(* CODESYS project 96lPixBadAppleControlWin.project

Project tree, tasks and I/O mapping:
  Device : CODESYS Control Win V3, 3S - Smart Software Solutions GmbH, order no. 305021, version 3.5.10.40
    application Application
      libraries: Standard, * (System); CAA File, 3.5.9.0 (CAA Technical Workgroup)
      task MainTask (cyclic, interval t#20ms, priority 1) calls PLC_PRG
      task VISU_TASK (cyclic, interval 100 ms, priority 31) calls VisuElems.Visu_Prg
      program PLC_PRG [ST]
      visualisation Visualization
      data type bigStruct
      data type bigUnion
      data type smallUnion
  visualisation LPixboard
  text list GlobalTextList
*)

// Device/Application/bigStruct
TYPE bigStruct :
STRUCT
	structLine0: ARRAY [0..11] OF BYTE;
	structLine1: ARRAY [0..11] OF BYTE;
	structLine2: ARRAY [0..11] OF BYTE;
	structLine3: ARRAY [0..11] OF BYTE;
	structLine4: ARRAY [0..11] OF BYTE;
	structLine5: ARRAY [0..11] OF BYTE;
	structLine6: ARRAY [0..11] OF BYTE;
	structLine7: ARRAY [0..11] OF BYTE;
	structLine8: ARRAY [0..11] OF BYTE;
	structLine9: ARRAY [0..11] OF BYTE;
	structLine10: ARRAY [0..11] OF BYTE;
	structLine11: ARRAY [0..11] OF BYTE;
	structLine12: ARRAY [0..11] OF BYTE;
	structLine13: ARRAY [0..11] OF BYTE;
	structLine14: ARRAY [0..11] OF BYTE;
	structLine15: ARRAY [0..11] OF BYTE;
	structLine16: ARRAY [0..11] OF BYTE;
	structLine17: ARRAY [0..11] OF BYTE;
	structLine18: ARRAY [0..11] OF BYTE;
	structLine19: ARRAY [0..11] OF BYTE;
	structLine20: ARRAY [0..11] OF BYTE;
	structLine21: ARRAY [0..11] OF BYTE;
	structLine22: ARRAY [0..11] OF BYTE;
	structLine23: ARRAY [0..11] OF BYTE;
	structLine24: ARRAY [0..11] OF BYTE;
	structLine25: ARRAY [0..11] OF BYTE;
	structLine26: ARRAY [0..11] OF BYTE;
	structLine27: ARRAY [0..11] OF BYTE;
	structLine28: ARRAY [0..11] OF BYTE;
	structLine29: ARRAY [0..11] OF BYTE;
	structLine30: ARRAY [0..11] OF BYTE;
	structLine31: ARRAY [0..11] OF BYTE;
	structLine32: ARRAY [0..11] OF BYTE;
	structLine33: ARRAY [0..11] OF BYTE;
	structLine34: ARRAY [0..11] OF BYTE;
	structLine35: ARRAY [0..11] OF BYTE;
	structLine36: ARRAY [0..11] OF BYTE;
	structLine37: ARRAY [0..11] OF BYTE;
	structLine38: ARRAY [0..11] OF BYTE;
	structLine39: ARRAY [0..11] OF BYTE;
	structLine40: ARRAY [0..11] OF BYTE;
	structLine41: ARRAY [0..11] OF BYTE;
	structLine42: ARRAY [0..11] OF BYTE;
	structLine43: ARRAY [0..11] OF BYTE;
	structLine44: ARRAY [0..11] OF BYTE;
	structLine45: ARRAY [0..11] OF BYTE;
	structLine46: ARRAY [0..11] OF BYTE;
	structLine47: ARRAY [0..11] OF BYTE;
	structLine48: ARRAY [0..11] OF BYTE;
	structLine49: ARRAY [0..11] OF BYTE;
	structLine50: ARRAY [0..11] OF BYTE;
	structLine51: ARRAY [0..11] OF BYTE;
	structLine52: ARRAY [0..11] OF BYTE;
	structLine53: ARRAY [0..11] OF BYTE;
	structLine54: ARRAY [0..11] OF BYTE;
	structLine55: ARRAY [0..11] OF BYTE;
	structLine56: ARRAY [0..11] OF BYTE;
	structLine57: ARRAY [0..11] OF BYTE;
	structLine58: ARRAY [0..11] OF BYTE;
	structLine59: ARRAY [0..11] OF BYTE;
	structLine60: ARRAY [0..11] OF BYTE;
	structLine61: ARRAY [0..11] OF BYTE;
	structLine62: ARRAY [0..11] OF BYTE;
	structLine63: ARRAY [0..11] OF BYTE;
	structLine64: ARRAY [0..11] OF BYTE;
	structLine65: ARRAY [0..11] OF BYTE;
	structLine66: ARRAY [0..11] OF BYTE;
	structLine67: ARRAY [0..11] OF BYTE;
	structLine68: ARRAY [0..11] OF BYTE;
	structLine69: ARRAY [0..11] OF BYTE;
	structLine70: ARRAY [0..11] OF BYTE;
	structLine71: ARRAY [0..11] OF BYTE;
END_STRUCT
END_TYPE

// Device/Application/bigUnion
TYPE bigUnion :
UNION
	pic: bigStruct;
	bigPic: ARRAY[0..863] OF BYTE;
END_UNION
END_TYPE

// Device/Application/smallUnion
TYPE smallUnion :
UNION
	bufferDWord: DWORD;
	bufferByte: ARRAY [0..3] OF BYTE;
END_UNION
END_TYPE

// Device/Application/PLC_PRG
PROGRAM PLC_PRG
VAR
	bigFrame0: bigUnion;
	
	matrix: ARRAY [0..863] OF BYTE;
	
	workStep: BYTE:= 0;
	
	trigDelay: TON;
	
	waitToStart: BOOL;
	
	fileOpen: FILE.Open;
	fileName: FILENAME:= 'e://project/fileName';
	fileOpenEn: BOOL;
	fileOpenDone: BOOL;
	fileHandle: __XWORD;
	
	fileRead: FILE.Read;
	fileBuffer: ARRAY[0..215] OF FILE.CAA.PVOID;
	fileBufferSize: UINT:= 864;
	fileReadEn: BOOL;
	
	fileClose: FILE.Close;
	fileCloseEn: BOOL;
	
	buffer: ARRAY[0..215] OF smallUnion;
	iFor: INT;
	iFourFor: INT;
	frameNo: DINT:= 0;
	frameNumbers: DINT:= 80000;
END_VAR

bigFrame0.bigPic:= matrix;

CASE workStep OF
	0:
		// wait click 'Start' button
		frameNo:= 0;
		IF waitToStart THEN
			workStep:= 1;
		END_IF
	1:
		// open the file
		fileOpenEn:= TRUE;
		IF fileHandle<>0 AND fileOpenDone THEN
			workStep:= 2;
		END_IF
	2:
		// read first Frame
		fileReadEn:= TRUE;
		IF fileRead.xDone THEN
			workStep:= 3;
		END_IF
	3:
		// close first read
		fileReadEn:= FALSE;
		IF NOT fileRead.xDone THEN
			workStep:= 4;
		END_IF
	4:
		// show this Frame
		FOR iFor:= 0 TO 215 BY 1 DO
			buffer[iFor].bufferDWord:= fileBuffer[iFor];
			FOR ifourFor:= 0 TO 3 BY 1 DO
				matrix[iFor*4 + iFourFor]:= buffer[iFor].bufferByte[iFourFor];
			END_FOR
		END_FOR
		IF iFor=216 THEN
			workStep:= 5;
		END_IF
	5:
		// frame delay
		frameNo:= frameNo + 1;
		trigDelay(IN:= TRUE, PT:= T#0.02S);
		IF trigDelay.Q THEN
			workStep:= 6;
		END_IF
	6:
		// close delay TON
		trigDelay(IN:= FALSE, PT:= T#0.02S);
		IF NOT trigDelay.Q THEN
			workStep:= 7;
		END_IF
	7:
		// check frame times
		IF frameNo<frameNumbers THEN
			workStep:= 2;
		END_IF
		IF frameNo>= frameNumbers THEN
			workStep:= 8;
		END_IF
	8:
		// close the file
		fileCloseEn:= TRUE;
		IF fileClose.xDone THEN
			workStep:= 9;
		END_IF
	9:
		// reset the FILE.Open FB
		fileOpenEn:= FALSE;
		IF NOT fileOpen.xDone THEN
			workStep:= 10;
		END_IF
	10:
		// reset the FILE.Close FB
		fileCloseEn:= FALSE;
		IF NOT fileClose.xDone THEN
			workStep:= 11;
		END_IF
END_CASE

fileOpen(sFileName:= fileName, eFileMode:= 1, xExclusive:= TRUE, xExecute:= fileOpenEn);
fileOpenDone:= fileOpen.xDone;

fileHandle:= fileOpen.hFile;

fileRead(hFile:= fileHandle, pBuffer:= ADR(fileBuffer), szBuffer:= fileBufferSize, xExecute:= fileReadEn);

fileClose(hFile:= fileHandle, xExecute:= fileCloseEn);

END_PROGRAM

// /LPixboard
VISUALIZATION LPixboard  // 194x4
VAR_IN_OUT
	pixArray: ARRAY[0..11] OF BYTE;
END_VAR
    Rectangle (0,0 2x2), invisible if: not pixArray[0].7
    Rectangle (2,0 2x2), invisible if: not pixArray[0].6
    Rectangle (4,0 2x2), invisible if: not pixArray[0].5
    Rectangle (6,0 2x2), invisible if: not pixArray[0].4
    Rectangle (8,0 2x2), invisible if: not pixArray[0].3
    Rectangle (10,0 2x2), invisible if: not pixArray[0].2
    Rectangle (12,0 2x2), invisible if: not pixArray[0].1
    Rectangle (14,0 2x2), invisible if: not pixArray[0].0
    Rectangle (16,0 2x2), invisible if: not pixArray[1].7
    Rectangle (18,0 2x2), invisible if: not pixArray[1].6
    Rectangle (20,0 2x2), invisible if: not pixArray[1].5
    Rectangle (22,0 2x2), invisible if: not pixArray[1].4
    Rectangle (24,0 2x2), invisible if: not pixArray[1].3
    Rectangle (26,0 2x2), invisible if: not pixArray[1].2
    Rectangle (28,0 2x2), invisible if: not pixArray[1].1
    Rectangle (30,0 2x2), invisible if: not pixArray[1].0
    Rectangle (32,0 2x2), invisible if: not pixArray[2].7
    Rectangle (34,0 2x2), invisible if: not pixArray[2].6
    Rectangle (36,0 2x2), invisible if: not pixArray[2].5
    Rectangle (38,0 2x2), invisible if: not pixArray[2].4
    Rectangle (40,0 2x2), invisible if: not pixArray[2].3
    Rectangle (42,0 2x2), invisible if: not pixArray[2].2
    Rectangle (44,0 2x2), invisible if: not pixArray[2].1
    Rectangle (46,0 2x2), invisible if: not pixArray[2].0
    Rectangle (48,0 2x2), invisible if: not pixArray[3].7
    Rectangle (50,0 2x2), invisible if: not pixArray[3].6
    Rectangle (52,0 2x2), invisible if: not pixArray[3].5
    Rectangle (54,0 2x2), invisible if: not pixArray[3].4
    Rectangle (56,0 2x2), invisible if: not pixArray[3].3
    Rectangle (58,0 2x2), invisible if: not pixArray[3].2
    Rectangle (60,0 2x2), invisible if: not pixArray[3].1
    Rectangle (62,0 2x2), invisible if: not pixArray[3].0
    Rectangle (64,0 2x2), invisible if: not pixArray[4].7
    Rectangle (66,0 2x2), invisible if: not pixArray[4].6
    Rectangle (68,0 2x2), invisible if: not pixArray[4].5
    Rectangle (70,0 2x2), invisible if: not pixArray[4].4
    Rectangle (72,0 2x2), invisible if: not pixArray[4].3
    Rectangle (74,0 2x2), invisible if: not pixArray[4].2
    Rectangle (76,0 2x2), invisible if: not pixArray[4].1
    Rectangle (78,0 2x2), invisible if: not pixArray[4].0
    Rectangle (80,0 2x2), invisible if: not pixArray[5].7
    Rectangle (82,0 2x2), invisible if: not pixArray[5].6
    Rectangle (84,0 2x2), invisible if: not pixArray[5].5
    Rectangle (86,0 2x2), invisible if: not pixArray[5].4
    Rectangle (88,0 2x2), invisible if: not pixArray[5].3
    Rectangle (90,0 2x2), invisible if: not pixArray[5].2
    Rectangle (92,0 2x2), invisible if: not pixArray[5].1
    Rectangle (94,0 2x2), invisible if: not pixArray[5].0
    Rectangle (96,0 2x2), invisible if: not pixArray[6].7
    Rectangle (98,0 2x2), invisible if: not pixArray[6].6
    Rectangle (100,0 2x2), invisible if: not pixArray[6].5
    Rectangle (102,0 2x2), invisible if: not pixArray[6].4
    Rectangle (104,0 2x2), invisible if: not pixArray[6].3
    Rectangle (106,0 2x2), invisible if: not pixArray[6].2
    Rectangle (108,0 2x2), invisible if: not pixArray[6].1
    Rectangle (110,0 2x2), invisible if: not pixArray[6].0
    Rectangle (112,0 2x2), invisible if: not pixArray[7].7
    Rectangle (114,0 2x2), invisible if: not pixArray[7].6
    Rectangle (116,0 2x2), invisible if: not pixArray[7].5
    Rectangle (118,0 2x2), invisible if: not pixArray[7].4
    Rectangle (120,0 2x2), invisible if: not pixArray[7].3
    Rectangle (122,0 2x2), invisible if: not pixArray[7].2
    Rectangle (124,0 2x2), invisible if: not pixArray[7].1
    Rectangle (126,0 2x2), invisible if: not pixArray[7].0
    Rectangle (128,0 2x2), invisible if: not pixArray[8].7
    Rectangle (130,0 2x2), invisible if: not pixArray[8].6
    Rectangle (132,0 2x2), invisible if: not pixArray[8].5
    Rectangle (134,0 2x2), invisible if: not pixArray[8].4
    Rectangle (136,0 2x2), invisible if: not pixArray[8].3
    Rectangle (138,0 2x2), invisible if: not pixArray[8].2
    Rectangle (140,0 2x2), invisible if: not pixArray[8].1
    Rectangle (142,0 2x2), invisible if: not pixArray[8].0
    Rectangle (144,0 2x2), invisible if: not pixArray[9].7
    Rectangle (146,0 2x2), invisible if: not pixArray[9].6
    Rectangle (148,0 2x2), invisible if: not pixArray[9].5
    Rectangle (150,0 2x2), invisible if: not pixArray[9].4
    Rectangle (152,0 2x2), invisible if: not pixArray[9].3
    Rectangle (154,0 2x2), invisible if: not pixArray[9].2
    Rectangle (156,0 2x2), invisible if: not pixArray[9].1
    Rectangle (158,0 2x2), invisible if: not pixArray[9].0
    Rectangle (160,0 2x2), invisible if: not pixArray[10].7
    Rectangle (162,0 2x2), invisible if: not pixArray[10].6
    Rectangle (164,0 2x2), invisible if: not pixArray[10].5
    Rectangle (166,0 2x2), invisible if: not pixArray[10].4
    Rectangle (168,0 2x2), invisible if: not pixArray[10].3
    Rectangle (170,0 2x2), invisible if: not pixArray[10].2
    Rectangle (172,0 2x2), invisible if: not pixArray[10].1
    Rectangle (174,0 2x2), invisible if: not pixArray[10].0
    Rectangle (176,0 2x2), invisible if: not pixArray[11].7
    Rectangle (178,0 2x2), invisible if: not pixArray[11].6
    Rectangle (180,0 2x2), invisible if: not pixArray[11].5
    Rectangle (182,0 2x2), invisible if: not pixArray[11].4
    Rectangle (184,0 2x2), invisible if: not pixArray[11].3
    Rectangle (186,0 2x2), invisible if: not pixArray[11].2
    Rectangle (188,0 2x2), invisible if: not pixArray[11].1
    Rectangle (190,0 2x2), invisible if: not pixArray[11].0
END_VISUALIZATION

// Device/Application/Visualization
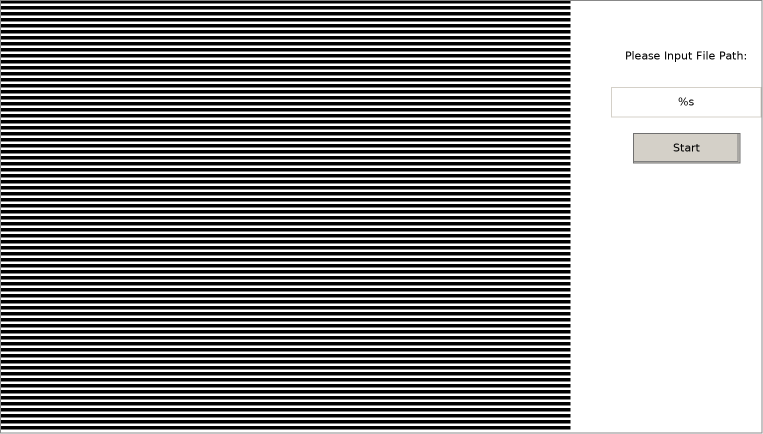
VISUALIZATION Visualization  // 763x434
    Frame (0,0 576x6)
        shows LPixboard(pixArray := PLC_PRG.bigFrame0.pic.structLine0)
    Frame (0,6 576x6)
        shows LPixboard(pixArray := PLC_PRG.bigFrame0.pic.structLine1)
    Frame (0,12 576x6)
        shows LPixboard(pixArray := PLC_PRG.bigFrame0.pic.structLine2)
    Frame (0,18 576x6)
        shows LPixboard(pixArray := PLC_PRG.bigFrame0.pic.structLine3)
    Frame (0,24 576x6)
        shows LPixboard(pixArray := PLC_PRG.bigFrame0.pic.structLine4)
    Frame (0,30 576x6)
        shows LPixboard(pixArray := PLC_PRG.bigFrame0.pic.structLine5)
    Frame (0,36 576x6)
        shows LPixboard(pixArray := PLC_PRG.bigFrame0.pic.structLine6)
    Frame (0,42 576x6)
        shows LPixboard(pixArray := PLC_PRG.bigFrame0.pic.structLine7)
    Frame (0,48 576x6)
        shows LPixboard(pixArray := PLC_PRG.bigFrame0.pic.structLine8)
    Frame (0,54 576x6)
        shows LPixboard(pixArray := PLC_PRG.bigFrame0.pic.structLine9)
    Frame (0,60 576x6)
        shows LPixboard(pixArray := PLC_PRG.bigFrame0.pic.structLine10)
    Frame (0,66 576x6)
        shows LPixboard(pixArray := PLC_PRG.bigFrame0.pic.structLine11)
    Frame (0,72 576x6)
        shows LPixboard(pixArray := PLC_PRG.bigFrame0.pic.structLine12)
    Frame (0,78 576x6)
        shows LPixboard(pixArray := PLC_PRG.bigFrame0.pic.structLine13)
    Frame (0,84 576x6)
        shows LPixboard(pixArray := PLC_PRG.bigFrame0.pic.structLine14)
    Frame (0,90 576x6)
        shows LPixboard(pixArray := PLC_PRG.bigFrame0.pic.structLine15)
    Frame (0,96 576x6)
        shows LPixboard(pixArray := PLC_PRG.bigFrame0.pic.structLine16)
    Frame (0,102 576x6)
        shows LPixboard(pixArray := PLC_PRG.bigFrame0.pic.structLine17)
    Frame (0,108 576x6)
        shows LPixboard(pixArray := PLC_PRG.bigFrame0.pic.structLine18)
    Frame (0,114 576x6)
        shows LPixboard(pixArray := PLC_PRG.bigFrame0.pic.structLine19)
    Frame (0,120 576x6)
        shows LPixboard(pixArray := PLC_PRG.bigFrame0.pic.structLine20)
    Frame (0,126 576x6)
        shows LPixboard(pixArray := PLC_PRG.bigFrame0.pic.structLine21)
    Frame (0,132 576x6)
        shows LPixboard(pixArray := PLC_PRG.bigFrame0.pic.structLine22)
    Frame (0,138 576x6)
        shows LPixboard(pixArray := PLC_PRG.bigFrame0.pic.structLine23)
    Frame (0,144 576x6)
        shows LPixboard(pixArray := PLC_PRG.bigFrame0.pic.structLine24)
    Frame (0,150 576x6)
        shows LPixboard(pixArray := PLC_PRG.bigFrame0.pic.structLine25)
    Frame (0,156 576x6)
        shows LPixboard(pixArray := PLC_PRG.bigFrame0.pic.structLine26)
    Frame (0,162 576x6)
        shows LPixboard(pixArray := PLC_PRG.bigFrame0.pic.structLine27)
    Frame (0,168 576x6)
        shows LPixboard(pixArray := PLC_PRG.bigFrame0.pic.structLine28)
    Frame (0,174 576x6)
        shows LPixboard(pixArray := PLC_PRG.bigFrame0.pic.structLine29)
    Frame (0,180 576x6)
        shows LPixboard(pixArray := PLC_PRG.bigFrame0.pic.structLine30)
    Frame (0,186 576x6)
        shows LPixboard(pixArray := PLC_PRG.bigFrame0.pic.structLine31)
    Frame (0,192 576x6)
        shows LPixboard(pixArray := PLC_PRG.bigFrame0.pic.structLine32)
    Frame (0,198 576x6)
        shows LPixboard(pixArray := PLC_PRG.bigFrame0.pic.structLine33)
    Frame (0,204 576x6)
        shows LPixboard(pixArray := PLC_PRG.bigFrame0.pic.structLine34)
    Frame (0,210 576x6)
        shows LPixboard(pixArray := PLC_PRG.bigFrame0.pic.structLine35)
    Frame (0,216 576x6)
        shows LPixboard(pixArray := PLC_PRG.bigFrame0.pic.structLine36)
    Frame (0,222 576x6)
        shows LPixboard(pixArray := PLC_PRG.bigFrame0.pic.structLine37)
    Frame (0,228 576x6)
        shows LPixboard(pixArray := PLC_PRG.bigFrame0.pic.structLine38)
    Frame (0,234 576x6)
        shows LPixboard(pixArray := PLC_PRG.bigFrame0.pic.structLine39)
    Frame (0,240 576x6)
        shows LPixboard(pixArray := PLC_PRG.bigFrame0.pic.structLine40)
    Frame (0,246 576x6)
        shows LPixboard(pixArray := PLC_PRG.bigFrame0.pic.structLine41)
    Frame (0,252 576x6)
        shows LPixboard(pixArray := PLC_PRG.bigFrame0.pic.structLine42)
    Frame (0,258 576x6)
        shows LPixboard(pixArray := PLC_PRG.bigFrame0.pic.structLine43)
    Frame (0,264 576x6)
        shows LPixboard(pixArray := PLC_PRG.bigFrame0.pic.structLine44)
    Frame (0,270 576x6)
        shows LPixboard(pixArray := PLC_PRG.bigFrame0.pic.structLine45)
    Frame (0,276 576x6)
        shows LPixboard(pixArray := PLC_PRG.bigFrame0.pic.structLine46)
    Frame (0,282 576x6)
        shows LPixboard(pixArray := PLC_PRG.bigFrame0.pic.structLine47)
    Frame (0,288 576x6)
        shows LPixboard(pixArray := PLC_PRG.bigFrame0.pic.structLine48)
    Frame (0,294 576x6)
        shows LPixboard(pixArray := PLC_PRG.bigFrame0.pic.structLine49)
    Frame (0,300 576x6)
        shows LPixboard(pixArray := PLC_PRG.bigFrame0.pic.structLine50)
    Frame (0,306 576x6)
        shows LPixboard(pixArray := PLC_PRG.bigFrame0.pic.structLine51)
    Frame (0,312 576x6)
        shows LPixboard(pixArray := PLC_PRG.bigFrame0.pic.structLine52)
    Frame (0,318 576x6)
        shows LPixboard(pixArray := PLC_PRG.bigFrame0.pic.structLine53)
    Frame (0,324 576x6)
        shows LPixboard(pixArray := PLC_PRG.bigFrame0.pic.structLine54)
    Frame (0,330 576x6)
        shows LPixboard(pixArray := PLC_PRG.bigFrame0.pic.structLine55)
    Frame (0,336 576x6)
        shows LPixboard(pixArray := PLC_PRG.bigFrame0.pic.structLine56)
    Frame (0,342 576x6)
        shows LPixboard(pixArray := PLC_PRG.bigFrame0.pic.structLine57)
    Frame (0,348 576x6)
        shows LPixboard(pixArray := PLC_PRG.bigFrame0.pic.structLine58)
    Frame (0,354 576x6)
        shows LPixboard(pixArray := PLC_PRG.bigFrame0.pic.structLine59)
    Frame (0,360 576x6)
        shows LPixboard(pixArray := PLC_PRG.bigFrame0.pic.structLine60)
    Frame (0,366 576x6)
        shows LPixboard(pixArray := PLC_PRG.bigFrame0.pic.structLine61)
    Frame (0,372 576x6)
        shows LPixboard(pixArray := PLC_PRG.bigFrame0.pic.structLine62)
    Frame (0,378 576x6)
        shows LPixboard(pixArray := PLC_PRG.bigFrame0.pic.structLine63)
    Frame (0,384 576x6)
        shows LPixboard(pixArray := PLC_PRG.bigFrame0.pic.structLine64)
    Frame (0,390 576x6)
        shows LPixboard(pixArray := PLC_PRG.bigFrame0.pic.structLine65)
    Frame (0,396 576x6)
        shows LPixboard(pixArray := PLC_PRG.bigFrame0.pic.structLine66)
    Frame (0,402 576x6)
        shows LPixboard(pixArray := PLC_PRG.bigFrame0.pic.structLine67)
    Frame (0,408 576x6)
        shows LPixboard(pixArray := PLC_PRG.bigFrame0.pic.structLine68)
    Frame (0,414 576x6)
        shows LPixboard(pixArray := PLC_PRG.bigFrame0.pic.structLine69)
    Frame (0,420 576x6)
        shows LPixboard(pixArray := PLC_PRG.bigFrame0.pic.structLine70)
    Frame (0,426 576x6)
        shows LPixboard(pixArray := PLC_PRG.bigFrame0.pic.structLine71)
    Textfield (611,87 150x30), "%s", text variable: PLC_PRG.fileName
        OnMouseClick: write the text variable via Edit
    Label (611,41 150x30), "Please Input File Path:"
    Button (633,133 107x30), "Start"
        tap PLC_PRG.waitToStart
END_VISUALIZATION
